(* LS Electric XG5000 project: 241002_실습3모터작동 *)
(* PLC LSPLC *)
(* module base 0 slot 0: 입력 모듈:XGI-D21A (DC 24V 입력, 8점 (전류소스/싱크입력)) *)
(* module base 0 slot 1: 출력 모듈:XGQ-RY1A (릴레이 출력, 8점 (2A용, 단독 COM.)) *)

PROGRAM NewProgram (* task: 스캔 프로그램 *)
VAR
    역방향버튼 AT %IX0.0.2 : BOOL;
    역방향으로회전 AT %QX0.1.1 : BOOL;
    정방향버튼 AT %IX0.0.1 : BOOL;
    정방향으로회전 AT %QX0.1.0 : BOOL;
    정지버튼 AT %IX0.0.3 : BOOL;
END_VAR

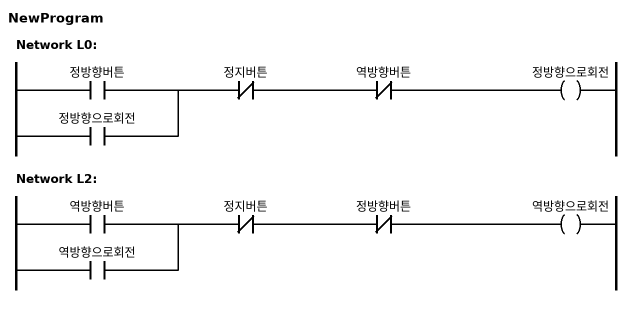
(* Rung L0 *)
정방향으로회전 := (정방향버튼 OR 정방향으로회전) AND NOT 정지버튼 AND NOT 역방향버튼;
(* Rung L2 *)
역방향으로회전 := (역방향버튼 OR 역방향으로회전) AND NOT 정지버튼 AND NOT 정방향버튼;
END_PROGRAM